{attribute 'GeneratedUsingTerminal: EL2252--0000'}
{attribute addProperty BoxType "EL2252--0000"}
{attribute addProperty Id "EtcSlaveTerminalBaseDC_Sync_ActivateAT %Q*DC_Sync_Activate_FA2D29101DC_Sync_StartAT %Q*DC_Sync_Start_9CCB0E514Channel_1AT %Q*Channel_42CA91F71Channel_2AT %Q*Channel_42CA91F71WcStateAT %I*WcState_0B2B16F91InfoDataAT %I*InfoData_A7436BC610"}
{attribute addProperty CRC "2037484372"}
{attribute addProperty Size "18"}
TYPE EL2252_79718B54 EXTENDS EtcSlaveTerminalBase :
STRUCT
	{attribute addProperty Name "DC_Sync_Activate"}
	DC_Sync_Activate : DC_Sync_Activate_FA2D2910;
	{attribute addProperty Name "DC_Sync_Start"}
	DC_Sync_Start : DC_Sync_Start_9CCB0E51;
	{attribute addProperty Name "Channel_1"}
	Channel_1 : Channel_42CA91F7;
	{attribute addProperty Name "Channel_2"}
	Channel_2 : Channel_42CA91F7;
	{attribute addProperty Name "WcState"}
	WcState : WcState_0B2B16F9;
	{attribute addProperty Name "InfoData"}
	InfoData : InfoData_A7436BC6;
END_STRUCT
END_TYPE

(* stored: Version 1.2.0.0, ProductVersion 3.1.4024.9
   DUT EL2252_79718B54: Id {9e5d7869-d004-403f-adc7-a288acdc845a} *)
